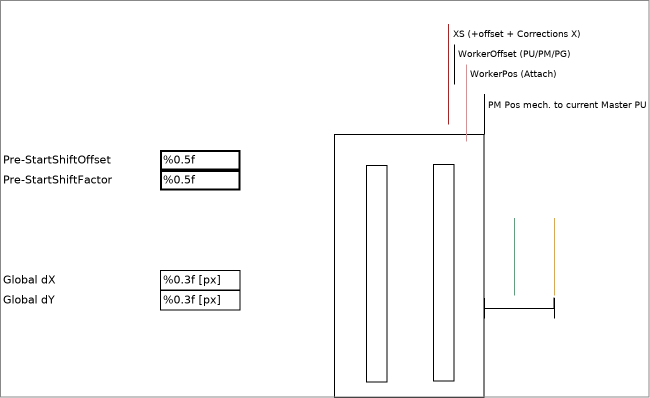
VISUALIZATION _VISU_WorkerDefGrid_Print_Pos  // 650x398
VAR_IN_OUT
  m_Inst : FB_WorkerDefGrid_Print;
END_VAR
    Rectangle (0,270 160x20), "Global dX"
    Rectangle (160,270 80x20), "%0.3f [px]", text variable: m_Inst._fDxGlobalShift
    Rectangle (0,290 160x20), "Global dY"
    Rectangle (160,290 80x20), "%0.3f [px]", text variable: m_Inst._fDyGlobalShift
    Rectangle (0,150 160x20), "Pre-StartShiftOffset"
    Rectangle (160,150 80x20), "%0.5f", text variable: m_Inst._fStartShiftOffset
        OnMouseDown: write the text variable via Default
    Rectangle (0,170 160x20), "Pre-StartShiftFactor"
    Rectangle (160,170 80x20), "%0.5f", text variable: m_Inst._fStartShiftFactor
        OnMouseDown: write the text variable via Default
    Rectangle (334,134 150x264)
    Group (481,94 6x40)
        Rectangle (0,0 6x40)
        Polyline (3,0) (3,40)
    RoundedRectangle (433,164 21x217)
    RoundedRectangle (366,165 21x217)
    Group (484,298 70x14)
        Rectangle (0,2 70x20)
        Polyline (0,0) (0,20) (0,10) (70,10) (70,0) (70,20)
    Group (451,44 6x120)
        Rectangle (0,0 6x40)
        Polyline (3,0) (3,40)
    Group (511,218 6x77)
        Rectangle (0,0 6x77)
        Polyline (3,0) (3,77)
    Group (551,218 6x77)
        Rectangle (0,0 6x77)
        Polyline (3,0) (3,77)
    Group (463,64 6x100)
        Rectangle (0,0 6x77)
        Polyline (3,0) (3,77)
    Rectangle (467,64 120x20), "WorkerPos (Attach)"
    Rectangle (485,95 165x20), "PM Pos mech. to current Master PU"
    Rectangle (455,44 130x20), "WorkerOffset (PU/PM/PG)"
    Group (445,24 6x140)
        Rectangle (0,0 6x100)
        Polyline (3,0) (3,100)
    Rectangle (450,24 130x20), "XS (+offset + Corrections X)"
END_VISUALIZATION

(* stored: Version 1.1.0.1, ProductVersion 3.1.4024.11
   Visu _VISU_WorkerDefGrid_Print_Pos: Id {95496a8f-15a7-4dbc-aed4-c2c751ade9cc} *)
